TYPE AdsTagsCTH2 :
STRUCT
	LA02: CTH_LA02;
END_STRUCT
END_TYPE

(* stored: Version 1.1.0.1, ProductVersion 3.1.4024.6
   DUT AdsTagsCTH2: Id {61ba002b-e1c2-450e-b09b-6530fd7327b7} *)
